INTERFACE I_DeserializerFeedback

METHOD PUBLIC LogError
VAR_INPUT
	Error : I_Error;
END_VAR
END_METHOD

END_INTERFACE

(* stored: Version 1.1.0.1, ProductVersion 3.1.4024.12
   Itf I_DeserializerFeedback: Id {3e85d5fa-0e05-0fac-2c00-bb2a66f70d26}
   Method LogError: Id {e5df8d5d-8a75-02cf-2818-217cc9cd3782} *)
